FUNCTION_BLOCK FB_RGBW
VAR_INPUT
	Betrieb			: BOOL;
	Farbcode	: STRING;
END_VAR
VAR_OUTPUT
END_VAR
VAR
	{attribute 'OPC.UA.DA' := '1'}Zustand			: ST_RGBW_Zustand;		
	{attribute 'OPC.UA.DA' := '1'}Steuerung		: ST_RGBW_Steuerung; 		
	Zustandscheck	: FB_RGBW_Zustandscheck;
END_VAR

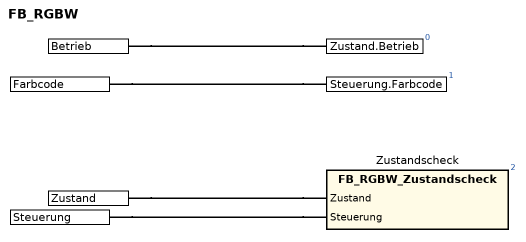
Zustand.Betrieb := Betrieb;
Steuerung.Farbcode := Farbcode;
Zustandscheck(Zustand := Zustand, Steuerung := Steuerung); // FB_RGBW_Zustandscheck

END_FUNCTION_BLOCK

(* stored: Version 1.1.0.1, ProductVersion 3.1.4024.9
   POU FB_RGBW: Id {b5f54a0d-e079-4103-a1a6-8adb82fe6492}, SpecialFunc None *)
